(* IEC 61131-3 sources: Temperature-control-using-fuzzy-logic/generated/plc, 1 file *)

(* ---- FB_FuzzyPIClimate.st ---- *)
(* Auto-generated by agriclimate.fuzzy.codegen - IEC 61131-3 Structured Text *)
(* Incremental fuzzy-PI climate controller. Call cyclically every tCycle.       *)
(* rDemand > 0 : heating demand, rDemand < 0 : cooling demand (-1 .. 1).        *)
FUNCTION_BLOCK FB_FuzzyPIClimate
VAR_INPUT
    rSetpoint   : REAL;          (* degC *)
    rMeasured   : REAL;          (* degC, validated sensor value *)
    rKe         : REAL := 0.3;   (* 1/degC  : error scaling *)
    rKr         : REAL := 200.0; (* s/degC  : error-rate scaling *)
    rKu         : REAL := 0.0015; (* 1/s     : output increment scaling *)
    rFilter     : REAL := 30.0;  (* s       : error-rate low-pass filter *)
    tCycle      : TIME := T#1S;
    xEnable     : BOOL;
    xTrack      : BOOL;          (* bumpless transfer: follow rTrackValue *)
    rTrackValue : REAL;
END_VAR
VAR_OUTPUT
    rDemand     : REAL;
END_VAR
VAR
    aLut   : ARRAY[0..440] OF REAL := [-0.8905, -0.8826, -0.8775, -0.8894, -0.8866, -0.8717, -0.8866, -0.8894, -0.8775, -0.8826, -0.8905, -0.7513, -0.6928, -0.6685, -0.5862, -0.5000, -0.4138, -0.2890, -0.1935, -0.1116, 0.0000, -0.8826, -0.8826, -0.8775, -0.8826, -0.8826, -0.8717, -0.8826, -0.8173, -0.7419, -0.7513, -0.7513, -0.6001, -0.5760, -0.5572, -0.4574, -0.3806, -0.3038, -0.1679, -0.0682, 0.0000, 0.1116, -0.8775, -0.8775, -0.8775, -0.8775, -0.8775, -0.8717, -0.8775, -0.8087, -0.7267, -0.6928, -0.6928, -0.5760, -0.5035, -0.4755, -0.3889, -0.3121, -0.2315, -0.0933, -0.0000, 0.0682, 0.1935, -0.8894, -0.8826, -0.8775, -0.8894, -0.8866, -0.8717, -0.8866, -0.8275, -0.7267, -0.6815, -0.6685, -0.5572, -0.4755, -0.3809, -0.2976, -0.2148, -0.1389, 0.0000, 0.0933, 0.1679, 0.2890, -0.8866, -0.8826, -0.8775, -0.8866, -0.7836, -0.7547, -0.7836, -0.7073, -0.6239, -0.5983, -0.5862, -0.4574, -0.3889, -0.2976, -0.1470, -0.0793, 0.0000, 0.1389, 0.2315, 0.3038, 0.4138, -0.8717, -0.8717, -0.8717, -0.8717, -0.7547, -0.7076, -0.7076, -0.6541, -0.5593, -0.5171, -0.5000, -0.3806, -0.3121, -0.2148, -0.0793, 0.0000, 0.0793, 0.2148, 0.3121, 0.3806, 0.5000, -0.8866, -0.8826, -0.8775, -0.8866, -0.7836, -0.7076, -0.6735, -0.6282, -0.5346, -0.4543, -0.4138, -0.3038, -0.2315, -0.1389, 0.0000, 0.0793, 0.1470, 0.2976, 0.3889, 0.4574, 0.5862, -0.8894, -0.8173, -0.8087, -0.8275, -0.7073, -0.6541, -0.6282, -0.5574, -0.4763, -0.3995, -0.2890, -0.1679, -0.0933, 0.0000, 0.1389, 0.2148, 0.2976, 0.3809, 0.4755, 0.5572, 0.6685, -0.8775, -0.7419, -0.7267, -0.7267, -0.6239, -0.5593, -0.5346, -0.4763, -0.3740, -0.3084, -0.1935, -0.0682, 0.0000, 0.0933, 0.2315, 0.3121, 0.3889, 0.4755, 0.5035, 0.5760, 0.6928, -0.8826, -0.7513, -0.6928, -0.6815, -0.5983, -0.5171, -0.4543, -0.3995, -0.3084, -0.2450, -0.1116, 0.0000, 0.0682, 0.1679, 0.3038, 0.3806, 0.4574, 0.5572, 0.5760, 0.6001, 0.7513, -0.8905, -0.7513, -0.6928, -0.6685, -0.5862, -0.5000, -0.4138, -0.2890, -0.1935, -0.1116, 0.0000, 0.1116, 0.1935, 0.2890, 0.4138, 0.5000, 0.5862, 0.6685, 0.6928, 0.7513, 0.8905, -0.7513, -0.6001, -0.5760, -0.5572, -0.4574, -0.3806, -0.3038, -0.1679, -0.0682, 0.0000, 0.1116, 0.2450, 0.3084, 0.3995, 0.4543, 0.5171, 0.5983, 0.6815, 0.6928, 0.7513, 0.8826, -0.6928, -0.5760, -0.5035, -0.4755, -0.3889, -0.3121, -0.2315, -0.0933, 0.0000, 0.0682, 0.1935, 0.3084, 0.3740, 0.4763, 0.5346, 0.5593, 0.6239, 0.7267, 0.7267, 0.7419, 0.8775, -0.6685, -0.5572, -0.4755, -0.3809, -0.2976, -0.2148, -0.1389, 0.0000, 0.0933, 0.1679, 0.2890, 0.3995, 0.4763, 0.5574, 0.6282, 0.6541, 0.7073, 0.8275, 0.8087, 0.8173, 0.8894, -0.5862, -0.4574, -0.3889, -0.2976, -0.1470, -0.0793, 0.0000, 0.1389, 0.2315, 0.3038, 0.4138, 0.4543, 0.5346, 0.6282, 0.6735, 0.7076, 0.7836, 0.8866, 0.8775, 0.8826, 0.8866, -0.5000, -0.3806, -0.3121, -0.2148, -0.0793, 0.0000, 0.0793, 0.2148, 0.3121, 0.3806, 0.5000, 0.5171, 0.5593, 0.6541, 0.7076, 0.7076, 0.7547, 0.8717, 0.8717, 0.8717, 0.8717, -0.4138, -0.3038, -0.2315, -0.1389, 0.0000, 0.0793, 0.1470, 0.2976, 0.3889, 0.4574, 0.5862, 0.5983, 0.6239, 0.7073, 0.7836, 0.7547, 0.7836, 0.8866, 0.8775, 0.8826, 0.8866, -0.2890, -0.1679, -0.0933, 0.0000, 0.1389, 0.2148, 0.2976, 0.3809, 0.4755, 0.5572, 0.6685, 0.6815, 0.7267, 0.8275, 0.8866, 0.8717, 0.8866, 0.8894, 0.8775, 0.8826, 0.8894, -0.1935, -0.0682, -0.0000, 0.0933, 0.2315, 0.3121, 0.3889, 0.4755, 0.5035, 0.5760, 0.6928, 0.6928, 0.7267, 0.8087, 0.8775, 0.8717, 0.8775, 0.8775, 0.8775, 0.8775, 0.8775, -0.1116, 0.0000, 0.0682, 0.1679, 0.3038, 0.3806, 0.4574, 0.5572, 0.5760, 0.6001, 0.7513, 0.7513, 0.7419, 0.8173, 0.8826, 0.8717, 0.8826, 0.8826, 0.8775, 0.8826, 0.8826, 0.0000, 0.1116, 0.1935, 0.2890, 0.4138, 0.5000, 0.5862, 0.6685, 0.6928, 0.7513, 0.8905, 0.8826, 0.8775, 0.8894, 0.8866, 0.8717, 0.8866, 0.8894, 0.8775, 0.8826, 0.8905];
    rErrPrev, rRateF, rE, rDe, rDu, rDt, fx, fy, rX, rY : REAL;
    ix, iy : INT;
    xInit  : BOOL;
END_VAR
VAR CONSTANT
    NX : INT := 21; NY : INT := 21;
    X0 : REAL := -1.0000; DX : REAL := 0.100000;
    Y0 : REAL := -1.0000; DY : REAL := 0.100000;
END_VAR

rDt := TIME_TO_REAL(tCycle) / 1000.0;
IF NOT xEnable THEN
    rDemand := 0.0; xInit := FALSE; RETURN;
END_IF
IF NOT xInit THEN
    rErrPrev := rSetpoint - rMeasured; rRateF := 0.0; xInit := TRUE;
END_IF
IF xTrack THEN
    rDemand := rTrackValue; rErrPrev := rSetpoint - rMeasured; RETURN;
END_IF

rE  := LIMIT(-1.0, (rSetpoint - rMeasured) * rKe, 1.0);
rRateF := rRateF + rDt / (rFilter + rDt) * (((rSetpoint - rMeasured) - rErrPrev) / rDt - rRateF);
rDe := LIMIT(-1.0, rRateF * rKr, 1.0);
rErrPrev := rSetpoint - rMeasured;

rX := (rE - X0) / DX;  rY := (rDe - Y0) / DY;
ix := MIN(REAL_TO_INT(TRUNC(rX)), NX - 2);  iy := MIN(REAL_TO_INT(TRUNC(rY)), NY - 2);
fx := rX - INT_TO_REAL(ix);  fy := rY - INT_TO_REAL(iy);
rDu := (1.0 - fx) * (1.0 - fy) * aLut[iy * NX + ix] + fx * (1.0 - fy) * aLut[iy * NX + ix + 1]
     + (1.0 - fx) * fy * aLut[(iy + 1) * NX + ix] + fx * fy * aLut[(iy + 1) * NX + ix + 1];

(* integrate with clamping anti-windup *)
rDemand := LIMIT(-1.0, rDemand + rKu * rDu * rDt, 1.0);
END_FUNCTION_BLOCK
